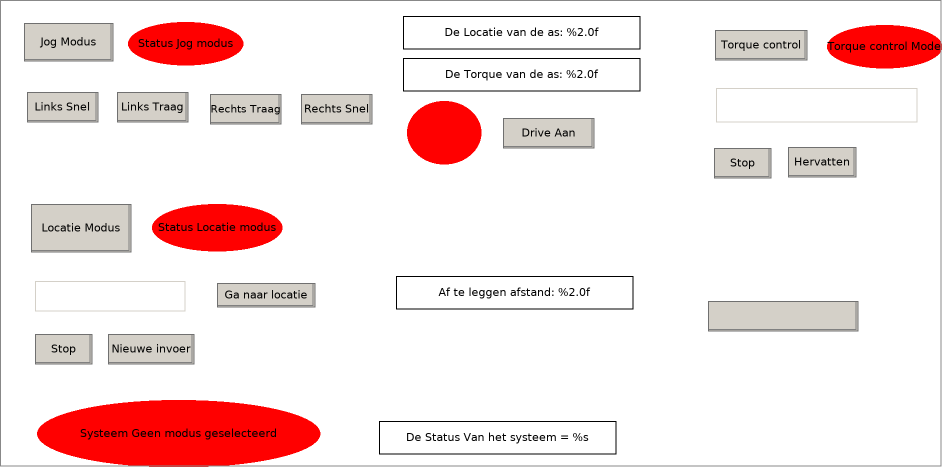
VISUALIZATION Visualization  // 942x467
    Button (503,118 91x30), "Drive Aan"
        toggle MAIN.CheckXas.KnopDriveAan2
    Ellipse (407,101 74x63), colour toggle: MAIN.CheckXas.IndicatieDriveIsActief
    Ellipse (128,22 115x43), "Status Jog modus", colour toggle: MAIN.CheckXas.IndicatieStatusIsJoggen
    Button (27,92 71x30), "Links Snel"
        tap MAIN.CheckXas.KnopJoggModusLinksSnel
    Button (117,92 71x30), "Links Traag"
        tap MAIN.CheckXas.KnopJoggModusLinksTraag
    Button (301,94 71x30), "Rechts Snel"
        tap MAIN.CheckXas.KnopJoggModusRechtsSnel
    Button (210,94 71x30), "Rechts Traag"
        tap MAIN.CheckXas.KnopJoggModusRechtsTraag
    Rectangle (403,16 237x33), "De Locatie van de as: %2.0f", text variable: MAIN.CheckXas.DePositieVanDeXas
    Textfield (35,281 150x30)
        OnMouseClick: write MAIN.CheckXas.DeIngevoerdeTargetPositie via VisuDialogs.Numpad
    Ellipse (152,204 130x47), "Status Locatie modus", colour toggle: MAIN.CheckXas.IndicatieStatusIsLocatie
    Button (217,283 98x24), "Ga naar locatie"
        tap MAIN.CheckXas.KnopLocatieUitvoeren
    Button (24,23 89x38), "Jog Modus"
        toggle MAIN.CheckXas.KnopJoggModus
    Button (31,204 100x48), "Locatie Modus"
        toggle MAIN.CheckXas.KnopLocatieModus
    Ellipse (37,400 283x67), "Systeem Geen modus geselecteerd", colour toggle: MAIN.CheckXas.IndicatieStatusIsUit
    Rectangle (396,276 237x33), "Af te leggen afstand: %2.0f", text variable: MAIN.CheckXas.NogAfTeLeggenAfstand
    Button (35,334 57x30), "Stop"
        tap MAIN.CheckXas.KnopStopKnop
    Button (108,334 86x30), "Nieuwe invoer"
        tap MAIN.CheckXas.KnopDoorgaan
    Button (715,30 92x30), "Torque control"
        toggle MAIN.CheckXas.KnopTorqueControl
    Ellipse (827,25 115x43), "Torque control Mode", colour toggle: MAIN.CheckXas.IndicatieStatusIsTorque
    Button (788,147 68x30), "Hervatten"
        tap MAIN.CheckXas.KnopHervatTorquecontrol
    Button (714,148 57x30), "Stop"
        tap MAIN.CheckXas.KnopStopKnop
    Textfield (716,88 201x34)
        OnMouseClick: write MAIN.CheckXas.DeIngevoerdeTorqueDoel via VisuDialogs.Numpad
    Button (708,301 150x30)
        tap MAIN.CheckXas.KnopSetPositionZero_Home
    Rectangle (403,58 237x33), "De Torque van de as: %2.0f", text variable: MAIN.CheckXas.DeTorqueVanDeXas
    Rectangle (379,421 237x33), "De Status Van het systeem = %s", text variable: MAIN.CheckXas.StatusVanDeStateVanHetSysteemText
END_VISUALIZATION

(* stored: Version 1.1.0.1, ProductVersion 3.1.4024.12
   Visu Visualization: Id {280b3afb-c641-4df6-8adf-14ddc99684bc} *)
